// TIA Portal V17 export
// export: Created 2024-08-29T18:23:50.5749143Z, ExportSetting WithDefaults, DisplayName Totally Integrated Automation Portal, DisplayVersion V17 Update 7, DisplayName TIA Portal Openness, DisplayVersion V17 Update 7, DisplayName TIA Portal Version Control Interface, DisplayVersion V17, DisplayName SINAMICS Startdrive Advanced, DisplayVersion V17 SP2, DisplayName SINAMICS Startdrive G110M, G120, G120C, G120D, G120P, G115D, DisplayVersion V17 SP2, DisplayName SINAMICS Startdrive G130, G150, S120, S150, SINAMICS MV, S210, DisplayVersion V17 SP2, DisplayName STEP 7 Professional, DisplayVersion V17 Update 7, DisplayName STEP 7 Safety, DisplayVersion V17 Update 6, DisplayName WinCC Advanced / Unified PC, DisplayVersion V17 Update 7
VAR_GLOBAL   // PLC tag table "HMIMemory"
   currentModel AT %MW3000 : Int;
   hmiButtonVisualization AT %M3050.6 : Bool;
   previousModel AT %MW3008 : Int;
   currentStep AT %MW3002 : Int;
   numberOfStepsToMove AT %MW3006 : UInt;
   stepToDivide AT %MW3012 : UInt;
   stepToInsert AT %MW3014 : UInt;
   hmiScreenNumber AT %MW3004 : Int;
   allowedTextChange AT %M3050.0 : Bool;
   progressBarMultiply AT %MW3010 : Int;
   lastCycleInputs AT %MD3034 : DInt;
   energySavingElapsedTime AT %MD3030 : Time;
   f7Button AT %M3050.5 : Bool;
   sequencerCopySequence AT %M3050.7 : Bool;
   codeReaderConfigurationVisible AT %M3050.2 : Bool;
   analogConfigurationVisible AT %M3050.1 : Bool;
   directAlarm AT %M3050.3 : Bool;
   directHome AT %M3050.4 : Bool;
   hmiRetractClampsReady AT %M3051.0 : Bool;
END_VAR
